// TIA Portal V17 export
// export: Created 2022-09-30T07:59:45.9762279Z, ExportSetting WithDefaults, DisplayName Totally Integrated Automation Portal, DisplayVersion V17 Update 5, DisplayName TIA Portal Openness, DisplayVersion V17 Update 5, DisplayName TIA Portal Teamcenter Gateway, DisplayVersion V17 Update 5, DisplayName TIA Portal Version Control Interface, DisplayVersion V17, DisplayName TIA Portal Test Suite Advanced, DisplayVersion V17 Update 1, DisplayName SINAMICS Startdrive Advanced, DisplayVersion V17 Update2, DisplayName SINAMICS Startdrive G130, G150, S120, S150, SINAMICS MV, S210, DisplayVersion V17 Update2, DisplayName SINAMICS Startdrive G110M, G120, G120C, G120D, G120P, G115D, DisplayVersion V17 Update2, DisplayName STEP 7 Professional, DisplayVersion V17 Update 5, DisplayName STEP 7 CFC, DisplayVersion V17 Update 1, DisplayName STEP 7 Safety, DisplayVersion V17, DisplayName WinCC Advanced / Unified PC, DisplayVersion V17 Update 5, DisplayName WinCC Unified Calendar, DisplayVersion V17, DisplayName WinCC Unified Performance Insight, DisplayVersion V17
TYPE "UDT_CALCUL"
// stored: IsFailsafeCompliant false
   STRUCT
      int_1 : Int;
      int_2 : Int;
      int_3 : Int;
      "Real" : Real;
      Result : Real;
   END_STRUCT;
END_TYPE
